{attribute 'OPC.UA.DA' := '1'}
FUNCTION_BLOCK Sapphire488Laser EXTENDS LaserBase
VAR_INPUT
END_VAR
VAR_OUTPUT
END_VAR
VAR
	{attribute 'OPC.UA.DA' := '0'}
	_config : Sapphire488LaserConfig;	
	{attribute 'OPC.UA.DA' := '0'}
	_coeAccess : CoeAccess;	
	{attribute 'OPC.UA.DA' := '0'}
	_initConfigSerialCom : BOOL;	
	{attribute 'OPC.UA.DA' := '0'}
	_suffix : STRING := Const.CR_LF;
	{attribute 'OPC.UA.DA' := '0'}
	_serialCom  : SerialCom(Prefix :='', Suffix := _suffix);
	{attribute 'OPC.UA.DA' := '0'}
	_refSerialCom : REFERENCE TO SerialCom(Prefix :='', Suffix := _suffix) := _serialCom;		 
	{attribute 'OPC.UA.DA' := '0'}
	_isReceived : BOOL;
	
	
	{attribute 'OPC.UA.DA' := '0'}
	_deliverMessages : INT;
	
	PowerMsg : STRING(255);
	InterlockStatusMsg : STRING(255);
	BasePlateTemperatureMsg : STRING(255);
	ControllerTemperatureMsg : STRING(255);
	DiodeSetTemperatureMsg : STRING(255);
	MeasuredTemperatureMsg : STRING(255);
	LaserHeadReachedDiodeCurrentLimitMsg : STRING(255);
	IdMsg : STRING(255);
	CustomMsg : STRING(255);
	
	{region 'Commands'}
	
	{attribute 'OPC.UA.DA' := '0'}
	_powerOn : BOOL;
	{attribute 'OPC.UA.DA' := '0'}
	_powerOff : BOOL;
	{attribute 'OPC.UA.DA' := '0'}
	_setPowerCmd : BOOL;
	{attribute 'OPC.UA.DA' := '0'}
	_customCmd : BOOL;	
	{attribute 'OPC.UA.DA' := '0'}			  		   
	_raiseProperties : BOOL;
	
	{endregion}			
	
	{attribute 'OPC.UA.DA' := '0'}
	_initDevice : BOOL;	
	 
	{attribute 'OPC.UA.DA' := '0'}
	_cmd : STRING;			
	{attribute 'OPC.UA.DA' := '0'}
	_setpoint : LREAL := 0;
	{attribute 'OPC.UA.DA' := '0'}
	_itemScheduler : INT;
	{attribute 'OPC.UA.DA' := '0'}
	_itemExecScheduler : INT;		
	{attribute 'OPC.UA.DA' := '0'}
	_itemRaisedProperties : INT;			
	{attribute 'OPC.UA.DA' := '0'}
	_pulseGenerator : TON;	
	{attribute 'OPC.UA.DA' := '0'}
	_execPulseGenerator : TON;	
			
	{attribute 'OPC.UA.DA' := '0'}
	fullMessage : STRING;
	{attribute 'OPC.UA.DA' := '0'}
	message : STRING;
	{attribute 'OPC.UA.DA' := '0'}	
	_length : INT;
	{attribute 'OPC.UA.DA' := '0'}	
	_suffixLength : INT := LEN(_suffix);	
END_VAR

IF NOT InitConfigSerialCom THEN
	ConfigureSerialCom();
ELSIF THIS^.Status = TExecutionState.Ready THEN
	IF _refSerialCom.ErrorReceiveId = COMERROR_NOERROR THEN
		_refSerialCom(TxBuffer:= HardwareGlobalVariables.TxBufferLaser, 
		 	      	  RxBuffer:= HardwareGlobalVariables.RxBufferLaser);
	END_IF				  
	
	// Init device
	IF NOT _initDevice THEN	
		InitDevice(); 		
	ELSE;
		// Deliver messages
		IF _refSerialCom.IsReceived THEN				 
			fullMessage := _refSerialCom.LastReceivedString;
			_length := LEN(fullMessage);
			message := DELETE(fullMessage, _suffixLength, _length-_suffixLength+1);
			
			CASE _deliverMessages OF			
				EFeedbackMsgSapphire488.PowerMsg :	
					PowerMsg := message;		
				EFeedbackMsgSapphire488.InterlockStatusMsg :
					InterlockStatusMsg := message;
				EFeedbackMsgSapphire488.BasePlateTemperatureMsg :
					BasePlateTemperatureMsg := message;
				EFeedbackMsgSapphire488.ControllerTemperatureMsg :
					ControllerTemperatureMsg := message;
				EFeedbackMsgSapphire488.DiodeSetTemperatureMsg :
					DiodeSetTemperatureMsg := message;
				EFeedbackMsgSapphire488.MeasuredTemperatureMsg :
					MeasuredTemperatureMsg := message;
				EFeedbackMsgSapphire488.LaserHeadReachedDiodeCurrentLimitMsg :
					LaserHeadReachedDiodeCurrentLimitMsg := message;
				EFeedbackMsgSapphire488.IdMsg :	
					IdMsg := message;
				EFeedbackMsgSapphire488.CustomMsg :
					CustomMsg := message;
			END_CASE		
		END_IF								   							   	
		
		PowerOn(_powerOn);
		PowerOff(_powerOff);	
		SetPower(_setPowerCmd, _setpoint);
		CustomCommand(_customCmd, _cmd);
		RaisePropertiesChanged(_raiseProperties);
		
		IF (NOT _powerOn AND NOT _powerOff AND NOT _setPowerCmd  
			AND NOT _customCmd AND NOT _raiseProperties) THEN
			MessageScheduler();
		END_IF
	
	END_IF
END_IF

METHOD ConfigureSerialCom
VAR_INPUT
END_VAR
IF _coeAccess.CoeOperation.Ready THEN
	_logger.Information(_message.Reset().Append('Start configuration com serial').ToString());
END_IF;	

_coeAccess.CoeOperation.Start();
_coeAccess(SerialCommunication := _config.SerialCommunication);
	
IF _coeAccess.CoeOperation.Done THEN
	_coeAccess.SetDone();	
	
	_Logger.Information(_message.Reset().
							Append('{').Append(TO_STRING(THIS^.Family)).Append('} : ').
							Append(' - Status : ').Append(TO_STRING(_coeAccess.Status)).ToString());	
	InitConfigSerialCom := TRUE;
END_IF
 
IF _coeAccess.CoeOperation.Error THEN	
	_coeAccess.SetError(0);
	
	_Logger.Error(_message.Reset().
							Append('{').Append(TO_STRING(THIS^.Family)).Append('} : ').
							Append(' - Status : ').Append(TO_STRING(_coeAccess.Status)).ToString());
	InitConfigSerialCom := TRUE;
END_IF

THIS^.Status := _coeAccess.Status;
State := _coeAccess.Status;
END_METHOD

{attribute 'TcRpcEnable' := '1'}
(** Custom command **)
METHOD CustomCommand
VAR_INPUT
	Execute : BOOL;
	Cmd : STRING;
END_VAR
IF Execute THEN
	_logger.Information(_message.Reset().
								Append(_config.Name).
								Append(' - Custom command : ').
								Append(Cmd).ToString());	
	_deliverMessages := EFeedbackMsgSapphire488.CustomMsg;														
	_serialCom.Send(Cmd);	
	_customCmd := FALSE;
END_IF
END_METHOD

METHOD FB_init : BOOL
VAR_INPUT
	bInitRetains : BOOL; // if TRUE, the retain variables are initialized (warm start / cold start)
	bInCopyCode : BOOL;  // if TRUE, the instance afterwards gets moved into the copy code (online change)
	Config : Sapphire488LaserConfig;
END_VAR
IF Config.IsEnabled THEN
	_config := Config;
	
	SUPER^._laserConfig.Name := Config.Name;
	SUPER^._laserConfig.DeviceID := Config.DeviceID;
	SUPER^._laserConfig.IsEnabled := Config.IsEnabled;
	SUPER^._laserConfig.LogLevel := Config.LogLevel;
	
	SUPER^.Name := Config.Name;
	SUPER^.DeviceID := Config.DeviceID;	
	THIS^.Family := DeviceFamily.Laser;
		
	_Logger.Information(_message.Reset().Append('Init ').
							Append('{').Append(TO_STRING(THIS^.Family)).Append('} - ').
							Append('{').Append(TO_STRING(Config.Name)).Append('}').ToString());																													
END_IF
END_METHOD

METHOD GetBasePlateTemperature 
VAR_INPUT
END_VAR
VAR
	cmd : STRING := '?BT';
END_VAR
_deliverMessages := EFeedbackMsgSapphire488.BasePlateTemperatureMsg;
_serialCom.Send(cmd);
END_METHOD

METHOD GetControllerTemperature
VAR_INPUT
END_VAR
VAR
	cmd : STRING := '?PST';
END_VAR
_deliverMessages := EFeedbackMsgSapphire488.ControllerTemperatureMsg;
_serialCom.Send(cmd);
END_METHOD

METHOD GetDiodeSetTemperature 
VAR_INPUT
END_VAR
VAR
	cmd : STRING := '?DST';
END_VAR
_deliverMessages := EFeedbackMsgSapphire488.DiodeSetTemperatureMsg;
_serialCom.Send(cmd);
END_METHOD

METHOD GetIdentifier
VAR_INPUT
END_VAR
VAR
	cmd : STRING := '?SV';
END_VAR
_deliverMessages := EFeedbackMsgSapphire488.IdMsg;
_serialCom.Send(cmd);
END_METHOD

(** Returns the status of the Interlock **)
METHOD PROTECTED GetInterlockStatus 
VAR_INPUT
END_VAR
VAR
	cmd : STRING := '?STA';
END_VAR
_deliverMessages := EFeedbackMsgSapphire488.InterlockStatusMsg;
_serialCom.Send(cmd);
END_METHOD

METHOD GetMeasuredTemperature 
VAR_INPUT
END_VAR
VAR
	cmd : STRING := '?DT';
END_VAR
_deliverMessages := EFeedbackMsgSapphire488.MeasuredTemperatureMsg;
_serialCom.Send(cmd);
END_METHOD

{attribute 'TcRpcEnable' := '1'}
(** Returns the timers of the laser and PSU:
		PSU Time=#######.#     Total time the system has been powered
		Laser Enabled Time=#######.#     Total time the diodes have been powered
		Laser OperationTime=#######.#    Total time the diodes have been powered >1 A  
**)
METHOD GetTimers : HoursStruct
VAR_INPUT
	Execute : BOOL;
END_VAR
VAR
	cmd : STRING := 'TIMERS?';
END_VAR
IF Execute THEN
	_logger.Information(_message.Reset().
								Append(_config.Name).
								Append(' - GetTimers').ToString());
	_serialCom.Send(cmd);
END_IF
END_METHOD

PROPERTY InitConfigSerialCom : BOOL
GET
InitConfigSerialCom := _initConfigSerialCom;
END_GET
SET
_initConfigSerialCom := InitConfigSerialCom;
END_SET
END_PROPERTY

METHOD InitDevice
VAR_INPUT
END_VAR
IF NOT _initDevice THEN	
	IF _pulseGenerator.Q THEN
		_pulseGenerator(IN := FALSE, PT := T#10MS);
			
		CASE _itemScheduler OF		
			0:	_logger.Information(_message.Reset().
								Append(_config.Name).
								Append(' - InitDevice').ToString());	

				_serialCom.Send('>=0'); // Echo off
				_itemScheduler := 1;				
		
			1:  _serialCom.Send('E=1'); // Set echo off
				_itemScheduler := 2;	
			
			2:  _serialCom.Send('T=1');  // Enable automatic servo regulation
				_itemScheduler := 3;	
    	
			3:	_raiseProperties:= TRUE;	
				_initDevice := TRUE;
				_itemScheduler := 0;
		END_CASE
	ELSE
	_pulseGenerator(IN := TRUE, PT := T#500MS);		
	END_IF
END_IF
END_METHOD

(** Returns the temperature of the laser head in degrees centigrade **)
METHOD LaserHeadReachedDiodeCurrentLimit 
VAR_INPUT
END_VAR
VAR
	cmd : STRING := '?MCR';
END_VAR
_deliverMessages := EFeedbackMsgSapphire488.LaserHeadReachedDiodeCurrentLimitMsg;
_serialCom.Send(cmd);
END_METHOD

METHOD MessageScheduler
VAR_INPUT
END_VAR
IF _pulseGenerator.Q THEN
	_pulseGenerator(IN := FALSE, PT := T#10MS);
		
	CASE _itemScheduler OF		
		0:	ReadPower();
			_itemScheduler := 1;				
	
		1:  GetBasePlateTemperature();
			_itemScheduler := 2;	
		
		2:  GetControllerTemperature();
			_itemScheduler := 3;		
			
		3:  GetDiodeSetTemperature();
			_itemScheduler := 4;
			
		4:  GetMeasuredTemperature();
			_itemScheduler := 5;
			
		5:  LaserHeadReachedDiodeCurrentLimit();
			_itemScheduler := 0;	
	END_CASE
ELSE
	_pulseGenerator(IN := TRUE, PT := T#500MS);		
END_IF
END_METHOD

{attribute 'TcRpcEnable' := '1'}
(** Disables the laser, regardless of the interlock status **)
METHOD PROTECTED PowerOff
VAR_INPUT
	Execute : BOOL;
END_VAR
VAR
	cmd : STRING := 'L=0';
END_VAR
IF Execute THEN	
	_powerOff := TRUE;	
	
	IF _execPulseGenerator.Q THEN
		_execPulseGenerator(IN := FALSE, PT := T#10MS);
			
		CASE _itemExecScheduler OF
			0: _logger.Information(_message.Reset().
								Append(_config.Name).
								Append(' - PowerOff').ToString());
				_serialCom.Send(cmd);
				_itemExecScheduler := 1;
			
			1:  GetInterlockStatus();
				_itemExecScheduler := 2;
				
			2:  _powerOff := FALSE;	
				_itemExecScheduler := 0;		
								
		END_CASE
	ELSE
		_execPulseGenerator(IN := TRUE, PT := T#500MS);	
	END_IF
END_IF
END_METHOD

{attribute 'TcRpcEnable' := '1'}
(* Enables the laser subject to Interlock and Enable Switch status *)
METHOD PROTECTED PowerOn
VAR_INPUT
	Execute : BOOL;
END_VAR
VAR
	cmd : STRING := 'L=1';
END_VAR
IF Execute THEN	
	_powerOn := TRUE;	

	IF _execPulseGenerator.Q THEN
		_execPulseGenerator(IN := FALSE, PT := T#10MS);
			
		CASE _itemExecScheduler OF
			0: _logger.Information(_message.Reset().
								Append(_config.Name).
								Append(' - PowerOn').ToString());
				_serialCom.Send(cmd);
				_itemExecScheduler := 1;
			
			1:  GetInterlockStatus();
				_itemExecScheduler := 2;
				
			2:  _powerOn := FALSE;	
				_itemExecScheduler := 0;		
								
		END_CASE
	ELSE
		_execPulseGenerator(IN := TRUE, PT := T#500MS);	
	END_IF
END_IF
END_METHOD

{attribute 'TcRpcEnable' := '1'}
METHOD RaisePropertiesChanged
VAR_INPUT
	Execute : BOOL;
END_VAR
IF Execute THEN
	_raiseProperties := TRUE;
	
	IF _pulseGenerator.Q THEN
		_pulseGenerator(IN := FALSE, PT := T#10MS);	

		CASE _itemRaisedProperties OF
			0:  InterlockStatusMsg := ' ';
				IdMsg := ' ';
				CustomMsg := ' ';
				
				_itemRaisedProperties := 10;
			
			10:  GetIdentifier();
				_itemRaisedProperties := 11;
				
			11:  GetInterlockStatus();
				_itemRaisedProperties := 12;
			
			12:  _logger.Information(_message.Reset().
								Append(_config.Name).
								Append(' - RaisePropertiesChanged').ToString());
				_raiseProperties := FALSE;				
				_itemRaisedProperties := 0;
			
		END_CASE
	ELSE
		_pulseGenerator(IN := TRUE, PT := T#500MS);	
	END_IF
END_IF
END_METHOD

(** Returns the power of the laser **)
METHOD PROTECTED ReadPower 
VAR_INPUT
END_VAR
VAR
	cmd : STRING := '?P';
END_VAR
_deliverMessages := EFeedbackMsgSapphire488.PowerMsg;	
_serialCom.Send(cmd);
END_METHOD

{attribute 'TcRpcEnable' := '1'}
(** This sets the output power of the laser 
For example, to set a power of 2800 mW, send the string POWER=2800, followed by striking the RETURN key
**)
METHOD PROTECTED SetPower 
VAR_INPUT
	Execute : BOOL;
	Power : LREAL;
END_VAR
VAR
	cmd : STRING := 'P=';
END_VAR
IF Execute THEN	
	_setPowerCmd := TRUE;	

	_setpoint := Power;
	
	IF _execPulseGenerator.Q THEN
		_execPulseGenerator(IN := FALSE, PT := T#10MS);
			
		CASE _itemExecScheduler OF
			0: _logger.Information(_message.Reset().
								Append(_config.Name).
								Append(' - SetPower : ').Append(TO_STRING(_setpoint)).ToString());
				_serialCom.Send(CONCAT(cmd, TO_STRING(_setpoint)));
				_itemExecScheduler := 1;
			
			1:  ReadPower();
				_itemExecScheduler := 2;
				
			2:  _setPowerCmd := FALSE;	
				_itemExecScheduler := 0;		
								
		END_CASE
	ELSE
		_execPulseGenerator(IN := TRUE, PT := T#500MS);	
	END_IF
END_IF
END_METHOD

END_FUNCTION_BLOCK

(* stored: Version 1.1.0.1, ProductVersion 3.1.4024.12
   POU Sapphire488Laser: Id {1b6d7450-4e40-4c5f-9193-3aaa5dd4ad37}, SpecialFunc None
   Folder Commands: Id {0d2596a8-7b7f-4860-9e21-e8b4ab5ebb69}
   Method ConfigureSerialCom: Id {5f2971b7-5cf9-47bf-a155-3c73b2e67abe}
   Method CustomCommand: Id {7e64e438-823c-472d-8a4f-2c03c9878109}
   Method FB_init: Id {f327e8ed-5d6d-4d5c-ae8e-eb5164770457}
   Method GetBasePlateTemperature: Id {01af3136-7314-4fa0-a7d7-2f2bd51213ac}
   Method GetControllerTemperature: Id {58f5886f-694a-48b1-b0e6-8bd1c2928280}
   Method GetDiodeSetTemperature: Id {ffb7c877-5a33-4e2f-9a0a-ba76d6513d51}
   Method GetIdentifier: Id {2c646a24-b2d1-47b0-aa96-bf539598d99d}
   Method GetInterlockStatus: Id {c581ed72-2540-4b2b-8880-4590bdf8a6bb}
   Method GetMeasuredTemperature: Id {b94b070d-4c93-49c2-a0cf-c5d640b165c1}
   Method GetTimers: Id {31c5ceb4-dbea-479c-b71f-e8b9133f5d45}
   Property InitConfigSerialCom: Id {4fe0c6d6-0a65-405b-8553-1f9f9045a6e0}
   Get Get: Id {8929ab3a-66d2-4d7f-b78f-c755c09f8a24}
   Set Set: Id {cc68e6c6-7caf-4573-9e6e-d63e573a5066}
   Method InitDevice: Id {6c49d82e-e1a8-48d9-ad3c-5dc801f9abf9}
   Method LaserHeadReachedDiodeCurrentLimit: Id {19b8cdbb-d8a9-4a22-ab0c-ab10aeac051b}
   Method MessageScheduler: Id {318fab93-b526-4999-816c-43d8686033b6}
   Method PowerOff: Id {44ab81af-7b5a-4400-9521-9722ed7b668f}
   Method PowerOn: Id {814f196c-0050-4a6f-9a8c-873d13d29ad1}
   Method RaisePropertiesChanged: Id {1ac4d013-b8b6-436a-a443-2a6f8f1db3a1}
   Method ReadPower: Id {b23b5f9f-66e0-4599-a78e-0774c9fc7296}
   Method SetPower: Id {bdd8421a-a68e-48d4-8053-66a148fdd0db} *)
